// TIA Portal V15.1 export
// export: Created 2024-06-21T08:41:10.0713844Z, ExportSetting WithDefaults, DisplayName Totally Integrated Automation Portal, DisplayVersion V15.1 Update 5, DisplayName TIA Portal Openness, DisplayVersion V15.1 Update 5, DisplayName SINAMICS Startdrive Advanced, DisplayVersion V15.1, DisplayName G130, G150, S120, S150, SINAMICS MV, S210, DisplayVersion V15.1, DisplayName G110M, G120, G120C, G120D, G120P, DisplayVersion V15.1, DisplayName STEP 7 Professional, DisplayVersion V15.1 Update 5, DisplayName STEP 7 Safety, DisplayVersion V15.1, DisplayName WinCC Professional, DisplayVersion V15.1 Update 5, DisplayName SIMATIC Visualization Architect, DisplayVersion V15.1
FUNCTION "LGBExtRol2W2S-MoviFitFCPN-Config" : Void   // FC6631, FBD
TITLE = LRoller2W2SG120PN-Config / LGBExtRol2W2S-MoviFitFCPN-Config
{ S7_Optimized_Access := 'TRUE' }
AUTHOR : ENGIE
FAMILY : Config
VERSION : 0.1
// =============================================================================
// Handles the LRoller2W2SG120PN Config
// =============================================================================
// ============================================================================
// Handles the LRoller2W2S-MoviFitFCPN Config
// ============================================================================
// stored: AutoNumber false, IsIECCheckEnabled false, SetENOAutomatically False, UDAEnableTagReadback false
   VAR_INPUT
      C_InitDirection : Bool;   // Config
      C_MotorProtectionNc : Bool;   // Config
      C_MotorProtectionUsed : Bool;   // Config
      C_MotionStopUsed : Bool;   // Config
      C_EnableAlarmHW : Bool;   // Enable Alarm hardware (e.g. safetyswitch, motorprotector, detections) / Config
      C_ReleaseBrakeUsed : Bool;   // Config
      C_NotQuickStop : Bool;   // Config
      C_Ramp : Time;   // Config
      C_ReferenceDriveCurrent : Real;   // Config
      C_ReferenceMotorCurrent : Real;   // Config
      C_ReferenceMotorRPM : Real;   // Config
      C_RatioGearbox : Real;   // Config
      C_Diameter : Real;   // Config
      C_Acceleration : Real;   // Config
      C_HWSubInput : HW_SUBMODULE;   // Config
      C_HWSubOutput : HW_SUBMODULE;   // Config
      C_HWSubInputStatus : HW_SUBMODULE;   // Config
   END_VAR
   VAR_IN_OUT
      IO_Config : "ExtRolConfig";   // Config
   END_VAR
BEGIN

REGION Network 1: **** 1 - Inputs **** Move Config
   // Move Config
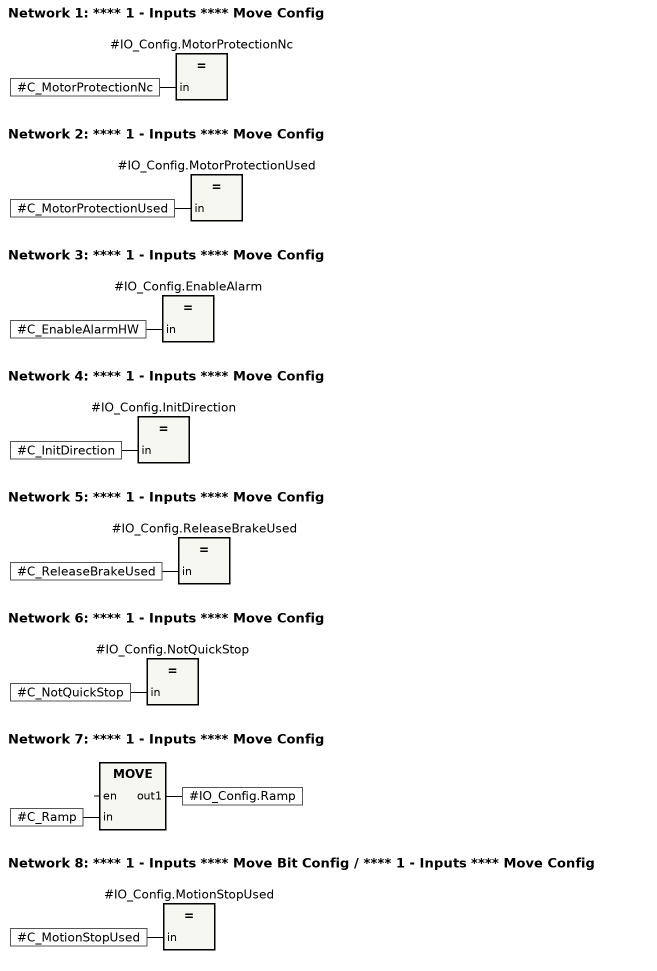
   #IO_Config.MotorProtectionNc := #C_MotorProtectionNc;
END_REGION

REGION Network 2: **** 1 - Inputs **** Move Config
   // Move Config
   #IO_Config.MotorProtectionUsed := #C_MotorProtectionUsed;
END_REGION

REGION Network 3: **** 1 - Inputs **** Move Config
   // Move Config
   #IO_Config.EnableAlarm := #C_EnableAlarmHW;
END_REGION

REGION Network 4: **** 1 - Inputs **** Move Config
   // Move Config
   #IO_Config.InitDirection := #C_InitDirection;
END_REGION

REGION Network 5: **** 1 - Inputs **** Move Config
   // Move Config
   #IO_Config.ReleaseBrakeUsed := #C_ReleaseBrakeUsed;
END_REGION

REGION Network 6: **** 1 - Inputs **** Move Config
   // Move Config
   #IO_Config.NotQuickStop := #C_NotQuickStop;
END_REGION

REGION Network 7: **** 1 - Inputs **** Move Config
   // Move Config
   #IO_Config.Ramp := #C_Ramp;
END_REGION

REGION Network 8: **** 1 - Inputs **** Move Bit Config / **** 1 - Inputs **** Move Config
   // Move Bit Config / Move Config
   #IO_Config.MotionStopUsed := #C_MotionStopUsed;
END_REGION

NETWORK
TITLE = **** 8 - Outputs **** Move Config UDT
// Move Config
      L     #C_ReferenceMotorCurrent;
      T     #IO_Config.ReferenceMotorCurrent;
      L     #C_ReferenceMotorRPM;
      T     #IO_Config.ReferenceMotorRPM;
      L     #C_RatioGearbox;
      T     #IO_Config.RatioGearbox;
      L     #C_Diameter;
      T     #IO_Config.Diameter;
      L     #C_Acceleration;
      T     #IO_Config.Acceleration;
      L     #C_ReferenceDriveCurrent;
      T     #IO_Config.ReferenceDriveCurrent;
      L     #C_HWSubInput;
      T     #IO_Config.HWSubInput;
      L     #C_HWSubOutput;
      T     #IO_Config.HWSubOutput;
      L     #C_HWSubInputStatus;
      T     #IO_Config.HWSubInputStatus;

END_FUNCTION
